// LS Electric XG5000 project: 동남118
// PLC NewPLC
// module base 0 slot 0: 입출력 모듈:XBC-DN/DP14E (DC 24V 입력 8점, 트랜지스터 출력 6점)

PROGRAM NewProgram (task: 스캔 프로그램)

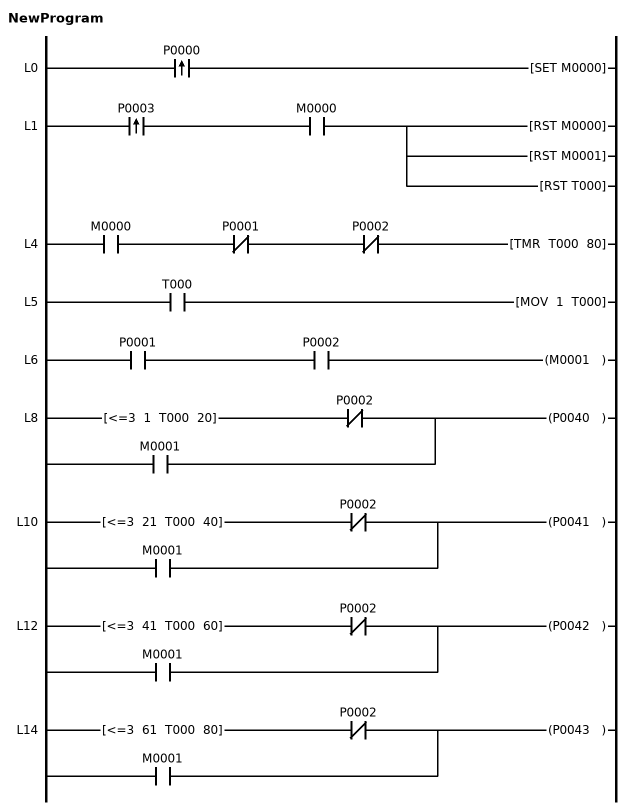
; L0
LOADP     P0000
SET       M0000
; L1
LOADP     P0003
AND       M0000
RST       M0000
RST       M0001
RST       T000
; L4
LOAD      M0000
AND NOT   P0001
AND NOT   P0002
TMR       T000 80
; L5
LOAD      T000
MOV       1 T000
; L6
LOAD      P0001
AND       P0002
OUT       M0001
; L8
LOAD<=3   1 T000 20
AND NOT   P0002
OR        M0001
OUT       P0040
; L10
LOAD<=3   21 T000 40
AND NOT   P0002
OR        M0001
OUT       P0041
; L12
LOAD<=3   41 T000 60
AND NOT   P0002
OR        M0001
OUT       P0042
; L14
LOAD<=3   61 T000 80
AND NOT   P0002
OR        M0001
OUT       P0043